// CheckRangeSigned checks subrange types of the type SINT, INT, DINT
// The purpose of this monitoring function is to deal with range bound violations as appropriate.
// Implicitly generated code : DO NOT EDIT
FUNCTION CheckRangeSigned : DINT
VAR_INPUT
	value, lower, upper: DINT;
END_VAR

// Implicitly generated code : Only an Implementation suggestion
{noflow}
IF (value < lower) THEN
	CheckRangeSigned := lower;
	GVL_TwinCatChecks.CheckRange_DINT_TooLow := GVL_TwinCatChecks.CheckRange_DINT_TooLow + 1;
ELSIF(value > upper) THEN
	CheckRangeSigned := upper;
	GVL_TwinCatChecks.CheckRange_DINT_TooHigh := GVL_TwinCatChecks.CheckRange_DINT_TooHigh + 1;
ELSE
	CheckRangeSigned := value;
END_IF
{flow}

END_FUNCTION

(* stored: Version 1.1.0.1, ProductVersion 3.1.4024.10
   POU CheckRangeSigned: Id {730f98ce-e8e6-4eba-9c6c-e9436fe418cd}, SpecialFunc CheckRangeSigned *)
